PROGRAM EM05_Placing4
VAR
	
	//Backbone
	FB_StateMachine_Placing4		: FB_StateManager;
	bFl_RunningMachinePlacing4		: BOOL;
	bFl_SeqReset					: BOOL;
	bFl_Manual						: BOOL;
	CheckStatusPlacing4				: checkstatus;
	AlarmEventHistory				: ARRAY[1..20] OF Alarm_Event_History;
	Placing4_Management				: FB_Placing_v2;
	bFl_Flushing					: BOOL;
	PalletID_Placing4				: PalletID_Name;
	Placing4_ID						: STRING;
	bFl_PalletJammed				: BOOL;
	
	//Motor
	Motor_PalletPlacing4			: MotorManagement;
	bFl_MotorPlacing4				: BOOL;
	Motor_Placing4_Error			: BOOL;
	Motor_Placing4_ErrorID			: UINT;
	bFl_MotorPlacing4_Fwd			: BOOL;
	bFl_MotorPlacing4_Rev			: BOOL;
	bFL_Safety						: BOOL;
	AlarmEventActive				: ARRAY[1..20] OF Alarm_Event_Active;
	CheckAcc						: TON;
END_VAR
VAR // added by the converter: edge detectors and wires of the graphical bodies
    _w1 : BOOL;
END_VAR

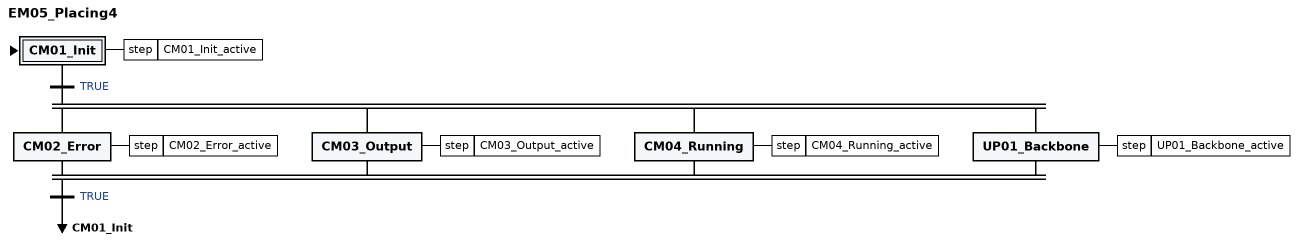
INITIAL_STEP CM01_Init:
    CM01_Init_active(N);  // step action
END_STEP
TRANSITION FROM CM01_Init TO (CM02_Error, CM03_Output, CM04_Running, UP01_Backbone)
    := TRUE;
END_TRANSITION
STEP CM02_Error:
    CM02_Error_active(N);  // step action
END_STEP
STEP CM03_Output:
    CM03_Output_active(N);  // step action
END_STEP
STEP CM04_Running:
    CM04_Running_active(N);  // step action
END_STEP
STEP UP01_Backbone:
    UP01_Backbone_active(N);  // step action
END_STEP
TRANSITION FROM (CM02_Error, CM03_Output, CM04_Running, UP01_Backbone) TO CM01_Init
    := TRUE;
END_TRANSITION

ACTION CM01_Init_active:
Data_GVL.bFL_StartPlacing4			:= Status_GVL.bFl_RunButton_Robotic OR HMI_GVL.bStartButtonPlacing4;
Data_GVL.bFL_StopPlacing4			:= NOT Status_GVL.bFl_StopButton_Robotic OR HMI_GVL.bStopButtonPlacing4;
Data_GVL.bFL_ResetPlacing4			:= Status_GVL.bFl_ResetButton_Robotic OR HMI_GVL.bResetButtonPlacing4;
Data_GVL.bFL_AckPlacing4			:= Status_GVL.bFl_Acknowledge_Robotic OR HMI_GVL.bAcknowledgeButtonPlacing4;
Data_GVL.bFL_AutoManuaModePlacing4 	:= Status_GVL.bFl_Manual_Robotic OR HMI_GVL.bTestModeEnablePlacing4;
bFl_RunningMachinePlacing4			:= Data_GVL.stStateMachinePlacing4.Running;
bFl_Manual							:= Data_GVL.stStateMachinePlacing4.ManualMode;
bFl_SeqReset						:= NOT Status_GVL.bFl_EStop_Robotic;
bFL_Safety							:= Status_GVL.bFl_EStop_Robotic AND Status_GVL.bSafety_DoorRobotic;



(*=================Convert Timer============================*)
Data_GVL.Tmr_Placing4	:= ConvertMilliSecTimeData(HMI_GVL.Tmr_Placing4);

(*=================Data OEE============================*)
Data_GVL.dt_Production[4].Data1			:= HMI_GVL.arCountTotal[4];
Data_GVL.dt_Production[4].Data2			:= HMI_GVL.arPalletTotal[4];
Data_GVL.dt_Production[4].Data3			:= HMI_GVL.arPalletIncomplete[4];
Data_GVL.dt_Production[4].ProductCode	:= Status_GVL.RecipeLine[4].ProductName;
END_ACTION

ACTION CM02_Error_active:
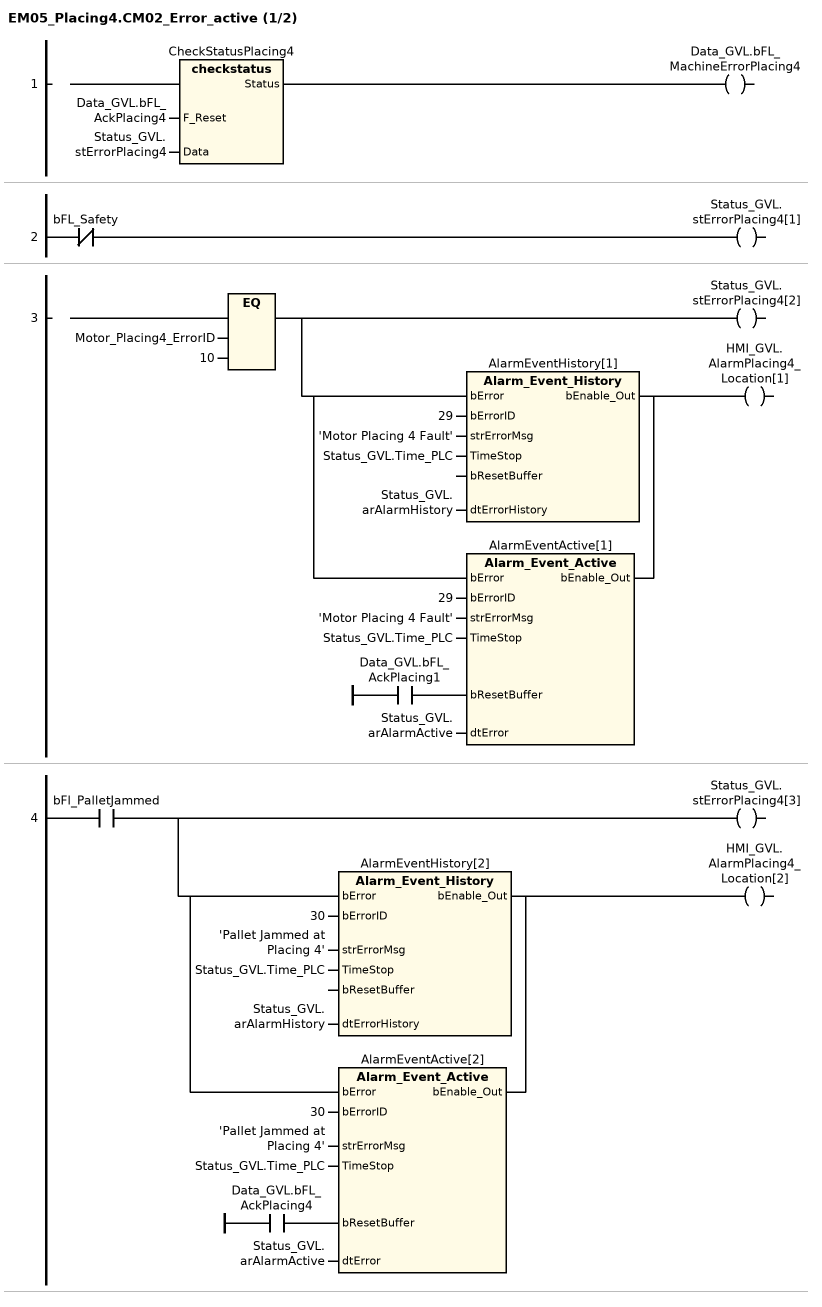
// NETWORK 1
CheckStatusPlacing4(F_Reset := Data_GVL.bFL_AckPlacing4, Data := Status_GVL.stErrorPlacing4); // checkstatus
Data_GVL.bFL_MachineErrorPlacing4 := CheckStatusPlacing4.Status;

// NETWORK 2
Status_GVL.stErrorPlacing4[1] := NOT bFL_Safety;

// NETWORK 3
_w1 := Motor_Placing4_ErrorID = 10;
Status_GVL.stErrorPlacing4[2] := _w1;
AlarmEventHistory[1](
    bError := _w1,
    bErrorID := 29,
    strErrorMsg := 'Motor Placing 4 Fault',
    TimeStop := Status_GVL.Time_PLC,
    dtErrorHistory := Status_GVL.arAlarmHistory); // Alarm_Event_History
AlarmEventActive[1](
    bError := _w1,
    bErrorID := 29,
    strErrorMsg := 'Motor Placing 4 Fault',
    TimeStop := Status_GVL.Time_PLC,
    bResetBuffer := Data_GVL.bFL_AckPlacing1,
    dtError := Status_GVL.arAlarmActive); // Alarm_Event_Active
HMI_GVL.AlarmPlacing4_Location[1] := AlarmEventHistory[1].bEnable_Out OR AlarmEventActive[1].bEnable_Out;

// NETWORK 4
Status_GVL.stErrorPlacing4[3] := bFl_PalletJammed;
AlarmEventHistory[2](
    bError := bFl_PalletJammed,
    bErrorID := 30,
    strErrorMsg := 'Pallet Jammed at Placing 4',
    TimeStop := Status_GVL.Time_PLC,
    dtErrorHistory := Status_GVL.arAlarmHistory); // Alarm_Event_History
AlarmEventActive[2](
    bError := bFl_PalletJammed,
    bErrorID := 30,
    strErrorMsg := 'Pallet Jammed at Placing 4',
    TimeStop := Status_GVL.Time_PLC,
    bResetBuffer := Data_GVL.bFL_AckPlacing4,
    dtError := Status_GVL.arAlarmActive); // Alarm_Event_Active
HMI_GVL.AlarmPlacing4_Location[2] := AlarmEventHistory[2].bEnable_Out OR AlarmEventActive[2].bEnable_Out;

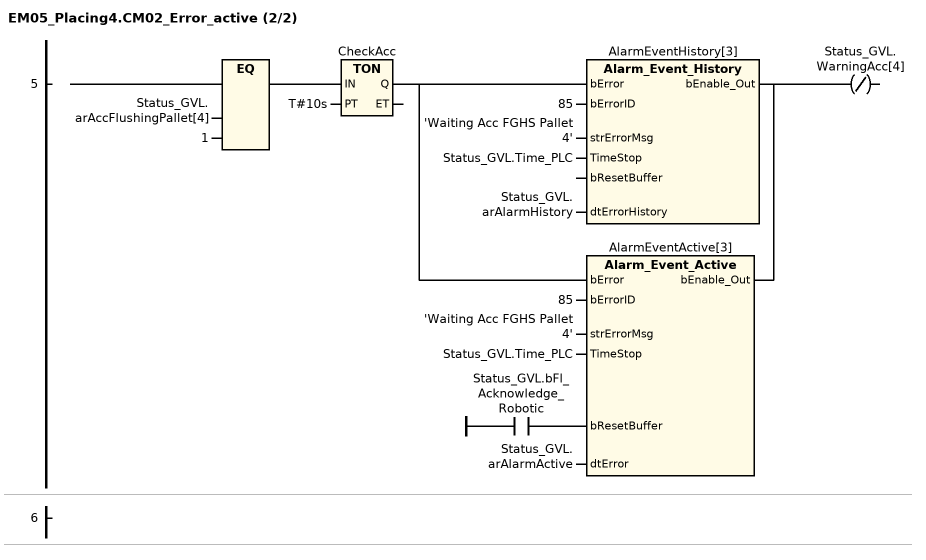
// NETWORK 5
CheckAcc(IN := Status_GVL.arAccFlushingPallet[4] = 1, PT := T#10s); // TON
AlarmEventHistory[3](
    bError := CheckAcc.Q,
    bErrorID := 85,
    strErrorMsg := 'Waiting Acc FGHS Pallet 4',
    TimeStop := Status_GVL.Time_PLC,
    dtErrorHistory := Status_GVL.arAlarmHistory); // Alarm_Event_History
AlarmEventActive[3](
    bError := CheckAcc.Q,
    bErrorID := 85,
    strErrorMsg := 'Waiting Acc FGHS Pallet 4',
    TimeStop := Status_GVL.Time_PLC,
    bResetBuffer := Status_GVL.bFl_Acknowledge_Robotic,
    dtError := Status_GVL.arAlarmActive); // Alarm_Event_Active
Status_GVL.WarningAcc[4] := NOT (AlarmEventHistory[3].bEnable_Out OR AlarmEventActive[3].bEnable_Out);

// NETWORK 6
END_ACTION

ACTION CM03_Output_active:
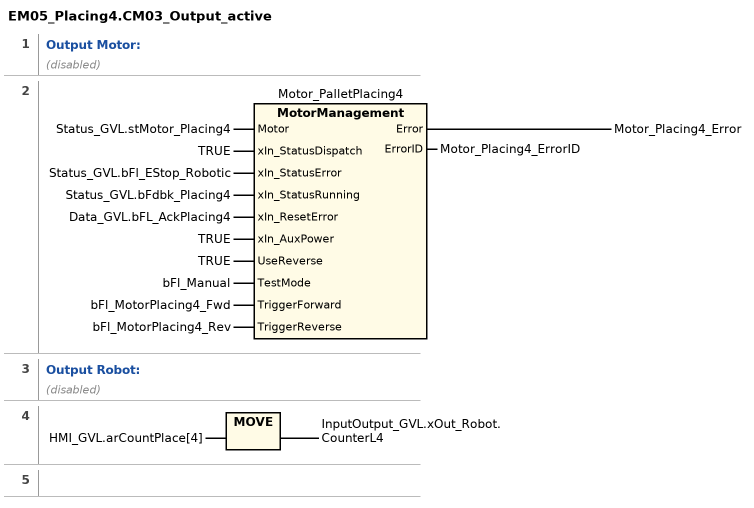
// NETWORK 1 (disabled)
// label: Output Motor

// NETWORK 2
Motor_PalletPlacing4(
    Motor := Status_GVL.stMotor_Placing4,
    xIn_StatusDispatch := TRUE,
    xIn_StatusError := Status_GVL.bFl_EStop_Robotic,
    xIn_StatusRunning := Status_GVL.bFdbk_Placing4,
    xIn_ResetError := Data_GVL.bFL_AckPlacing4,
    xIn_AuxPower := TRUE,
    UseReverse := TRUE,
    TestMode := bFl_Manual,
    TriggerForward := bFl_MotorPlacing4_Fwd,
    TriggerReverse := bFl_MotorPlacing4_Rev,
    ErrorID => Motor_Placing4_ErrorID); // MotorManagement
Motor_Placing4_Error := Motor_PalletPlacing4.Error;

// NETWORK 3 (disabled)
// label: Output Robot

// NETWORK 4
InputOutput_GVL.xOut_Robot.CounterL4 := HMI_GVL.arCountPlace[4];

// NETWORK 5
END_ACTION

ACTION CM04_Running_active:
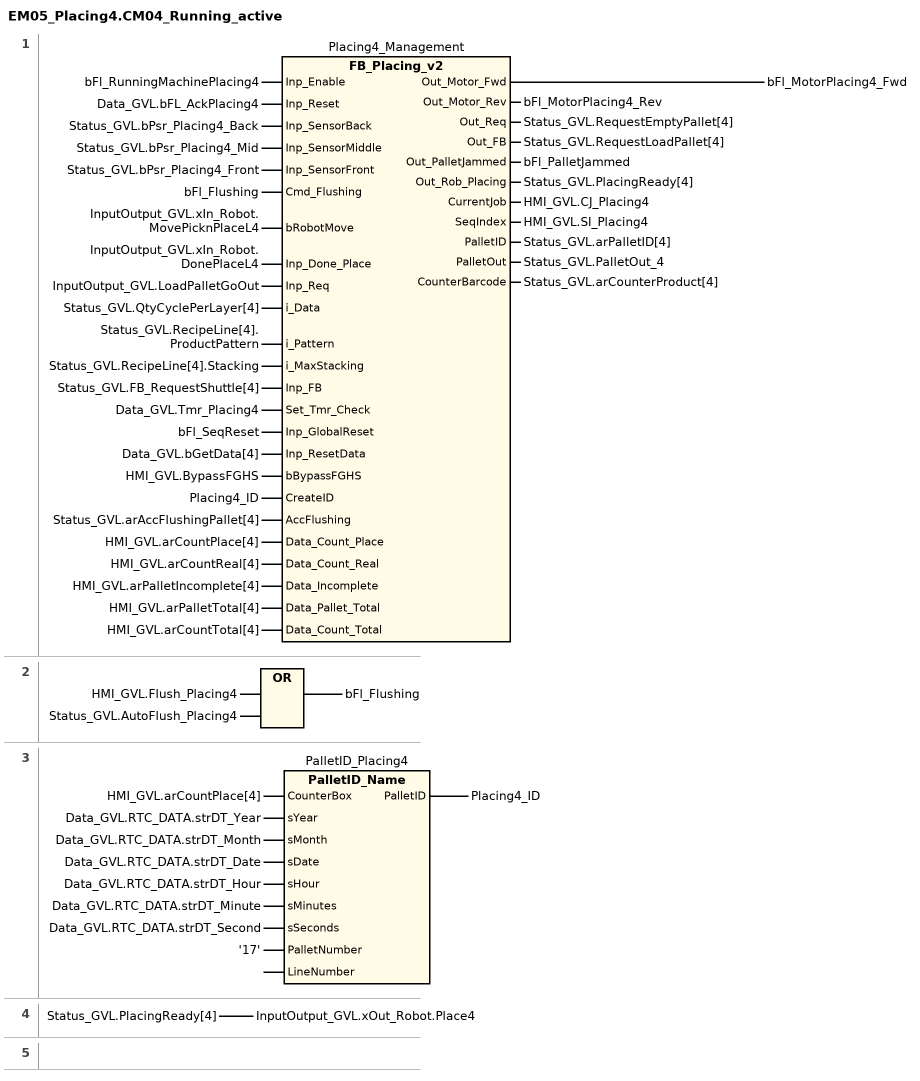
// NETWORK 1
Placing4_Management(
    Inp_Enable := bFl_RunningMachinePlacing4,
    Inp_Reset := Data_GVL.bFL_AckPlacing4,
    Inp_SensorBack := Status_GVL.bPsr_Placing4_Back,
    Inp_SensorMiddle := Status_GVL.bPsr_Placing4_Mid,
    Inp_SensorFront := Status_GVL.bPsr_Placing4_Front,
    Cmd_Flushing := bFl_Flushing,
    bRobotMove := InputOutput_GVL.xIn_Robot.MovePicknPlaceL4,
    Inp_Done_Place := InputOutput_GVL.xIn_Robot.DonePlaceL4,
    Inp_Req := InputOutput_GVL.LoadPalletGoOut,
    i_Data := Status_GVL.QtyCyclePerLayer[4],
    i_Pattern := Status_GVL.RecipeLine[4].ProductPattern,
    i_MaxStacking := Status_GVL.RecipeLine[4].Stacking,
    Inp_FB := Status_GVL.FB_RequestShuttle[4],
    Set_Tmr_Check := Data_GVL.Tmr_Placing4,
    Inp_GlobalReset := bFl_SeqReset,
    Inp_ResetData := Data_GVL.bGetData[4],
    bBypassFGHS := HMI_GVL.BypassFGHS,
    CreateID := Placing4_ID,
    AccFlushing := Status_GVL.arAccFlushingPallet[4],
    Data_Count_Place := HMI_GVL.arCountPlace[4],
    Data_Count_Real := HMI_GVL.arCountReal[4],
    Data_Incomplete := HMI_GVL.arPalletIncomplete[4],
    Data_Pallet_Total := HMI_GVL.arPalletTotal[4],
    Data_Count_Total := HMI_GVL.arCountTotal[4],
    Out_Motor_Rev => bFl_MotorPlacing4_Rev,
    Out_Req => Status_GVL.RequestEmptyPallet[4],
    Out_FB => Status_GVL.RequestLoadPallet[4],
    Out_PalletJammed => bFl_PalletJammed,
    Out_Rob_Placing => Status_GVL.PlacingReady[4],
    CurrentJob => HMI_GVL.CJ_Placing4,
    SeqIndex => HMI_GVL.SI_Placing4,
    PalletID => Status_GVL.arPalletID[4],
    PalletOut => Status_GVL.PalletOut_4,
    CounterBarcode => Status_GVL.arCounterProduct[4]); // FB_Placing_v2
bFl_MotorPlacing4_Fwd := Placing4_Management.Out_Motor_Fwd;

// NETWORK 2
bFl_Flushing := HMI_GVL.Flush_Placing4 OR Status_GVL.AutoFlush_Placing4;

// NETWORK 3
PalletID_Placing4(
    CounterBox := HMI_GVL.arCountPlace[4],
    sYear := Data_GVL.RTC_DATA.strDT_Year,
    sMonth := Data_GVL.RTC_DATA.strDT_Month,
    sDate := Data_GVL.RTC_DATA.strDT_Date,
    sHour := Data_GVL.RTC_DATA.strDT_Hour,
    sMinutes := Data_GVL.RTC_DATA.strDT_Minute,
    sSeconds := Data_GVL.RTC_DATA.strDT_Second,
    PalletNumber := '17'); // PalletID_Name
Placing4_ID := PalletID_Placing4.PalletID;

// NETWORK 4
InputOutput_GVL.xOut_Robot.Place4 := Status_GVL.PlacingReady[4];

// NETWORK 5
END_ACTION

ACTION UP01_Backbone_active:
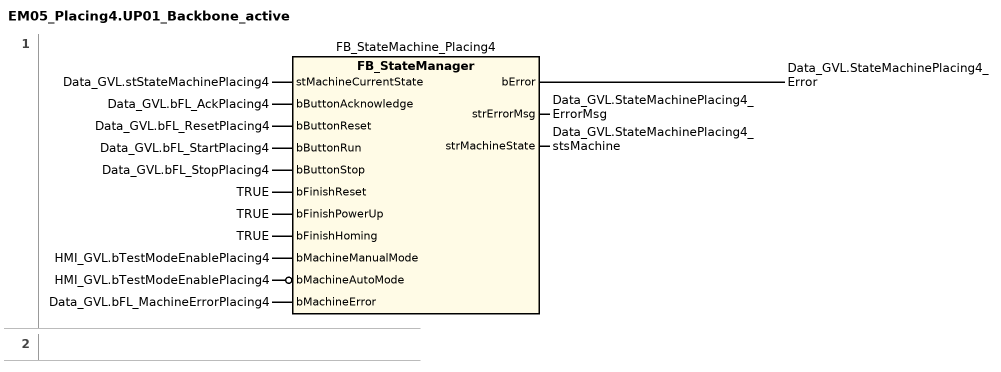
// NETWORK 1
FB_StateMachine_Placing4(
    stMachineCurrentState := Data_GVL.stStateMachinePlacing4,
    bButtonAcknowledge := Data_GVL.bFL_AckPlacing4,
    bButtonReset := Data_GVL.bFL_ResetPlacing4,
    bButtonRun := Data_GVL.bFL_StartPlacing4,
    bButtonStop := Data_GVL.bFL_StopPlacing4,
    bFinishReset := TRUE,
    bFinishPowerUp := TRUE,
    bFinishHoming := TRUE,
    bMachineManualMode := HMI_GVL.bTestModeEnablePlacing4,
    bMachineAutoMode := NOT HMI_GVL.bTestModeEnablePlacing4,
    bMachineError := Data_GVL.bFL_MachineErrorPlacing4,
    strErrorMsg => Data_GVL.StateMachinePlacing4_ErrorMsg,
    strMachineState => Data_GVL.StateMachinePlacing4_stsMachine); // FB_StateManager
Data_GVL.StateMachinePlacing4_Error := FB_StateMachine_Placing4.bError;

// NETWORK 2
END_ACTION

END_PROGRAM

(* stored: Version 1.1.0.1, ProductVersion 3.1.4024.12
   POU EM05_Placing4: Id {f73a8ed5-259f-4269-a1fd-20ac3f3cec23}, SpecialFunc None
   Action CM01_Init_active: Id {6258c882-7f31-476c-a458-5901cccd2ba0}
   Action CM02_Error_active: Id {de878d67-f356-4f34-a8e4-b3081765971d}
   Action CM03_Output_active: Id {1c21b3b1-402d-4a16-b3e8-9b384604e3dd}
   Action CM04_Running_active: Id {b9b3d491-ace5-46ef-8d29-ea3d63907cc6}
   Action UP01_Backbone_active: Id {e57dff52-8868-4e3d-bb50-f700092f0c95} *)
